PROGRAM MAIN
VAR
	fbLongRunning		: TON := (PT:=T#4s);
	counter				: UINT;
	fbTof: TOF;
END_VAR

Commands.StartCommand1.Call();

fbTof(
	IN := Commands.StartCommand1.Q,
	PT := T#1S);
	





counter := counter + 1;


// Function variant
Commands.AddCommand1.Call();
Commands.DelayedAddCommand1.Call();

// Strukture variant
IF Commands.stAddCommand.stCmd.bExecute THEN
	Commands.stAddCommand.stArgsOut.result :=
		Commands.stAddCommand.stArgsIn.a + Commands.stAddCommand.stArgsIn.b;
	Commands.stAddCommand.stCmd.nResultCode := 0;
	Commands.stAddCommand.stCmd.bBusy := Commands.stAddCommand.stCmd.bExecute := FALSE;
END_IF

// Länger gehendes Kommando
IF Commands.stAddLongCommand.stCmd.bExecute THEN
	Commands.stAddLongCommand.stCmd.bBusy := TRUE;
END_IF

IF NOT Commands.stAddLongCommand.stCmd.bExecute AND Commands.stAddLongCommand.stCmd.bBusy THEN
	Commands.stAddLongCommand.stCmd.bBusy := FALSE;
	Commands.stAddLongCommand.stCmd.nResultCode := 5;
END_IF

fbLongRunning(IN:=Commands.stAddLongCommand.stCmd.bBusy);

IF fbLongRunning.Q THEN
	Commands.stAddLongCommand.stArgsOut.result :=
		Commands.stAddLongCommand.stArgsIn.a + Commands.stAddLongCommand.stArgsIn.b;
	Commands.stAddLongCommand.stCmd.nResultCode := 0;
	Commands.stAddLongCommand.stCmd.bBusy := Commands.stAddLongCommand.stCmd.bExecute := FALSE;	
END_IF

END_PROGRAM

(* stored: Version 1.1.0.1, ProductVersion 3.1.4022.10
   POU MAIN: Id {12ac386e-9f2f-456d-9446-322109fb7ee0}, SpecialFunc None *)
